{attribute 'GeneratedUsingTerminal: EK1100-0000-0018'}
{attribute addProperty BoxType "EK1100-0000-0018"}
{attribute addProperty Id "Beckhoff_ELM37xxEK1122Beckhoff_ELM37xxEK1122_E40DDF852A_0001_ELM3702_0000_0016ELM3702_3D4ED79F42A_0002_ELM3702_0000_0017ELM3702_3D4ED79F42A_0003_ELM3704_0000_0016ELM3704_177D76D464A_0004_ELM3704_0000_0017ELM3704_177D76D464A_0005_ELM3704_0001_0017ELM3704_177D76D464A_0006_ELM3704_0020_0016ELM3704_177D76D464A_0007_ELM3702_0101_0016ELM3702_3D4ED79F42A_0008_ELM3704_1001_0016ELM3704_177D76D464A_0009_ELM3704_1001_0017ELM3704_177D76D464"}
{attribute addProperty CRC "1476565822"}
{attribute addProperty Size "512"}
TYPE Beckhoff_ELM37xx_58029B3E EXTENDS EK1100_1FC0878B :
STRUCT
	{attribute addProperty Name "Beckhoff_ELM37xxEK1122"}
	{attribute addProperty PreviousPort "Beckhoff ELM37xx : B"}
	Beckhoff_ELM37xxEK1122 : Beckhoff_ELM37xxEK1122_E40DDF85;
	{attribute addProperty Name "A_0001_ELM3702_0000_0016"}
	{attribute addProperty PreviousPort "Beckhoff ELM37xxEK1122 : C"}
	A_0001_ELM3702_0000_0016 : ELM3702_3D4ED79F;
	{attribute addProperty Name "A_0002_ELM3702_0000_0017"}
	{attribute addProperty PreviousPort "A_0001(ELM3702-0000-0016) : B"}
	A_0002_ELM3702_0000_0017 : ELM3702_3D4ED79F;
	{attribute addProperty Name "A_0003_ELM3704_0000_0016"}
	{attribute addProperty PreviousPort "A_0002(ELM3702-0000-0017) : B"}
	A_0003_ELM3704_0000_0016 : ELM3704_177D76D4;
	{attribute addProperty Name "A_0004_ELM3704_0000_0017"}
	{attribute addProperty PreviousPort "A_0003(ELM3704-0000-0016) : B"}
	A_0004_ELM3704_0000_0017 : ELM3704_177D76D4;
	{attribute addProperty Name "A_0005_ELM3704_0001_0017"}
	{attribute addProperty PreviousPort "A_0004(ELM3704-0000-0017) : B"}
	A_0005_ELM3704_0001_0017 : ELM3704_177D76D4;
	{attribute addProperty Name "A_0006_ELM3704_0020_0016"}
	{attribute addProperty PreviousPort "A_0005(ELM3704-0001-0017) : B"}
	A_0006_ELM3704_0020_0016 : ELM3704_177D76D4;
	{attribute addProperty Name "A_0007_ELM3702_0101_0016"}
	{attribute addProperty PreviousPort "A_0006(ELM3704-0020-0016) : B"}
	A_0007_ELM3702_0101_0016 : ELM3702_3D4ED79F;
	{attribute addProperty Name "A_0008_ELM3704_1001_0016"}
	{attribute addProperty PreviousPort "A_0007(ELM3702-0101-0016) : B"}
	A_0008_ELM3704_1001_0016 : ELM3704_177D76D4;
	{attribute addProperty Name "A_0009_ELM3704_1001_0017"}
	{attribute addProperty PreviousPort "A_0008(ELM3704-1001-0016) : B"}
	A_0009_ELM3704_1001_0017 : ELM3704_177D76D4;
END_STRUCT
END_TYPE

(* stored: Version 1.2.0.0, ProductVersion 3.1.4024.9
   DUT Beckhoff_ELM37xx_58029B3E: Id {6d6c6654-26a6-410f-9d93-dc04098b5d59} *)
